Staubli VAL3: clearScreen.pgx

public program clearScreen()
begin

  // Clear pendant screen

  cls(scMonitor)

end
